// TIA Portal V18 export
// export: Created 2026-01-09T11:32:03.26758Z, ExportSetting WithDefaults, DisplayName Totally Integrated Automation Portal, DisplayVersion V18 Update 5, DisplayName TIA Portal Openness, DisplayVersion V18 Update 5, DisplayName TIA Portal Teamcenter Gateway, DisplayVersion V18, DisplayName TIA Portal Version Control Interface, DisplayVersion V18, DisplayName SINAMICS Startdrive Advanced, DisplayVersion V18 SP2 Update 1, DisplayName SINAMICS Startdrive G110M, G120, G120C, G120D, G120P, G115D, DisplayVersion V18 SP2 Update 1, DisplayName SINAMICS Startdrive G130, G150, S120, S150, SINAMICS MV, S210, G220, S200, DisplayVersion V18 SP2 Update 1, DisplayName STEP 7 Professional, DisplayVersion V18 Update 5, DisplayName STEP 7 Safety, DisplayVersion V18, DisplayName WinCC Professional, DisplayVersion V18 Update 5
TagTable "U"
  _UserName : WString  (1 s)
  _UserLevel : Int  (1 s)
  _unlock : Array [0..9] of Bool  (1 s)
    TagArrayMember "[0]"
    TagArrayMember "[1]"
    TagArrayMember "[2]"
    TagArrayMember "[3]"
    TagArrayMember "[4]"
    TagArrayMember "[5]"
    TagArrayMember "[6]"
    TagArrayMember "[7]"
    TagArrayMember "[8]"
    TagArrayMember "[9]"
